// TIA Portal V17 export
// export: Created 2023-02-13T11:16:22.5513855Z, ExportSetting WithDefaults, DisplayName Totally Integrated Automation Portal, DisplayVersion V17, DisplayName TIA Portal Openness, DisplayVersion V17, DisplayName TIA Portal Teamcenter Gateway, DisplayVersion V17, DisplayName TIA Portal Version Control Interface, DisplayVersion V17, DisplayName SINAMICS Startdrive Advanced, DisplayVersion V17, DisplayName SINAMICS Startdrive G130, G150, S120, S150, SINAMICS MV, S210, DisplayVersion V17, DisplayName SINAMICS Startdrive G110M, G120, G120C, G120D, G120P, G115D, DisplayVersion V17, DisplayName STEP 7 Professional, DisplayVersion V17, DisplayName STEP 7 Safety, DisplayVersion V17, DisplayName WinCC Professional, DisplayVersion V17
DATA_BLOCK "IO_Valve_Blend40_DB"   // DB26
VERSION : 0.1
// stored: AutoNumber true, DBAccessibleFromOPCUA true, DBAccessibleFromWebserver true, InstanceOfName IO_Valve_Blend40, InstanceOfType FB
"IO_Valve_Blend40"
   // VAR_INPUT
   //    "lock 1" : Bool;
   //    "lock 2" : Bool;
   //    "lock 3" : Bool;
   //    "lock 4" : Bool;
   //    init : Bool;
   //    reset : Bool;
   //    testing : Bool;
   // END_VAR
   // VAR
   //    "AV-40.01" : "Valve";
   //    "AV-40.02" : "Valve";
   //    "AV-40.03" : "Valve";
   //    "AV-40.04" : "Valve";
   //    "AV-40.05" : "Valve";
   //    "AV-40.06" : "Valve";
   //    "AV-40.07" : "Valve";
   //    "AV-40.08" : "Valve";
   //    "AV-40.09" : "Valve";
   //    "AV-40.10" : "Valve";
   //    "AV-40.11" : "Valve";
   //    "AV-40.21" : "Valve";
   //    "AV-40.22" : "Valve";
   //    "AV-40.23" : "Valve";
   //    "AV-40.24" : "Valve";
   //    "AV-40.25" : "Valve";
   //    "AV-40.26" : "Valve";
   //    "AV-40.27" : "Valve";
   //    "AV-40.28" : "Valve";
   //    "AV-40.29" : "Valve";
   //    "AV-40.30" : "Valve";
   //    "AV-40.31" : "Valve";
   //    "AV-40.32" : "Valve";
   //    "AV-40.33" : "Valve";
   //    "AV-40.34" : "Valve";
   // END_VAR
BEGIN
END_DATA_BLOCK
